// TIA Portal V18 export
// export: Created 2026-03-12T16:04:32.2344065Z, ExportSetting WithDefaults, DisplayName Totally Integrated Automation Portal, DisplayVersion V18 Update 5, DisplayName TIA Portal Openness, DisplayVersion V18 Update 5, DisplayName TIA Portal Version Control Interface, DisplayVersion V18, DisplayName SINAMICS Startdrive Advanced, DisplayVersion V18, DisplayName SINAMICS Startdrive G130, G150, S120, S150, SINAMICS MV, S210, DisplayVersion V18, DisplayName SINAMICS Startdrive G110M, G120, G120C, G120D, G120P, G115D, DisplayVersion V18, DisplayName STEP 7 Professional, DisplayVersion V18 Update 5, DisplayName STEP 7 Safety, DisplayVersion V18, DisplayName WinCC Professional, DisplayVersion V18 Update 5
ORGANIZATION_BLOCK "Main"   // OB1, LAD, ProgramCycle
TITLE = "Main Program Sweep (Cycle)"
{ S7_Optimized_Access := 'TRUE' }
VERSION : 0.1
// Este bloco verifica as condições dos sinais discretos dos painéis. Se as condições operacionais não forem atendidas, as FCs respectivas de cada painel são intertravadas no item 2. Fluxo de Controle.
// stored: AutoNumber true, IsIECCheckEnabled false, SetENOAutomatically false
   VAR_INPUT
      Initial_Call : Bool;   // Initial call of this OB
      Remanence : Bool;   // =True, if remanent data are available
   END_VAR
BEGIN

REGION Network 1: Intertravamento Painel CCO
   // Se o Botão de Emergência estiver Desacionado Painel CCO OK
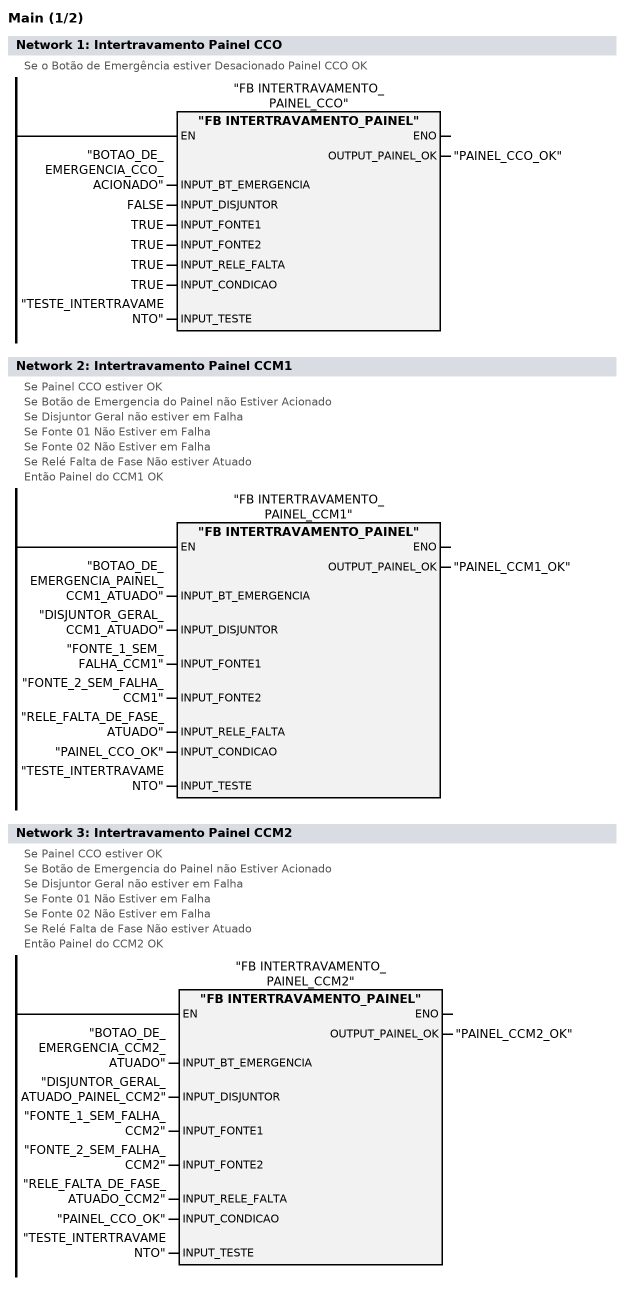
   RUNG wire#powerrail
      "FB INTERTRAVAMENTO_PAINEL_CCO"(INPUT_BT_EMERGENCIA := "BOTAO_DE_EMERGENCIA_CCO_ACIONADO", INPUT_DISJUNTOR := FALSE, INPUT_FONTE1 := TRUE, INPUT_FONTE2 := TRUE, INPUT_RELE_FALTA := TRUE, INPUT_CONDICAO := TRUE, INPUT_TESTE := "TESTE_INTERTRAVAMENTO", OUTPUT_PAINEL_OK => "PAINEL_CCO_OK")
   END_RUNG
   // the same network as SCL:
   "FB INTERTRAVAMENTO_PAINEL_CCO"(INPUT_BT_EMERGENCIA := "BOTAO_DE_EMERGENCIA_CCO_ACIONADO",   // "FB INTERTRAVAMENTO_PAINEL"
                           INPUT_DISJUNTOR := FALSE,
                           INPUT_FONTE1 := TRUE,
                           INPUT_FONTE2 := TRUE,
                           INPUT_RELE_FALTA := TRUE,
                           INPUT_CONDICAO := TRUE,
                           INPUT_TESTE := "TESTE_INTERTRAVAMENTO",
                           OUTPUT_PAINEL_OK => "PAINEL_CCO_OK");
END_REGION

REGION Network 2: Intertravamento Painel CCM1
   // Se Painel CCO estiver OK
   // Se Botão de Emergencia do Painel não Estiver Acionado
   // Se Disjuntor Geral não estiver em Falha
   // Se Fonte 01 Não Estiver em Falha
   // Se Fonte 02 Não Estiver em Falha
   // Se Relé Falta de Fase Não estiver Atuado
   // Então Painel do CCM1 OK
   RUNG wire#powerrail
      "FB INTERTRAVAMENTO_PAINEL_CCM1"(INPUT_BT_EMERGENCIA := "BOTAO_DE_EMERGENCIA_PAINEL_CCM1_ATUADO", INPUT_DISJUNTOR := "DISJUNTOR_GERAL_CCM1_ATUADO", INPUT_FONTE1 := "FONTE_1_SEM_ FALHA_CCM1", INPUT_FONTE2 := "FONTE_2_SEM_FALHA_CCM1", INPUT_RELE_FALTA := "RELE_FALTA_DE_FASE_ATUADO", INPUT_CONDICAO := "PAINEL_CCO_OK", INPUT_TESTE := "TESTE_INTERTRAVAMENTO", OUTPUT_PAINEL_OK => "PAINEL_CCM1_OK")
   END_RUNG
   // the same network as SCL:
   "FB INTERTRAVAMENTO_PAINEL_CCM1"(INPUT_BT_EMERGENCIA := "BOTAO_DE_EMERGENCIA_PAINEL_CCM1_ATUADO",   // "FB INTERTRAVAMENTO_PAINEL"
                           INPUT_DISJUNTOR := "DISJUNTOR_GERAL_CCM1_ATUADO",
                           INPUT_FONTE1 := "FONTE_1_SEM_ FALHA_CCM1",
                           INPUT_FONTE2 := "FONTE_2_SEM_FALHA_CCM1",
                           INPUT_RELE_FALTA := "RELE_FALTA_DE_FASE_ATUADO",
                           INPUT_CONDICAO := "PAINEL_CCO_OK",
                           INPUT_TESTE := "TESTE_INTERTRAVAMENTO",
                           OUTPUT_PAINEL_OK => "PAINEL_CCM1_OK");
END_REGION

REGION Network 3: Intertravamento Painel CCM2
   // Se Painel CCO estiver OK
   // Se Botão de Emergencia do Painel não Estiver Acionado
   // Se Disjuntor Geral não estiver em Falha
   // Se Fonte 01 Não Estiver em Falha
   // Se Fonte 02 Não Estiver em Falha
   // Se Relé Falta de Fase Não estiver Atuado
   // Então Painel do CCM2 OK
   RUNG wire#powerrail
      "FB INTERTRAVAMENTO_PAINEL_CCM2"(INPUT_BT_EMERGENCIA := "BOTAO_DE_EMERGENCIA_CCM2_ATUADO", INPUT_DISJUNTOR := "DISJUNTOR_GERAL_ATUADO_PAINEL_CCM2", INPUT_FONTE1 := "FONTE_1_SEM_FALHA_CCM2", INPUT_FONTE2 := "FONTE_2_SEM_FALHA_CCM2", INPUT_RELE_FALTA := "RELE_FALTA_DE_FASE_ATUADO_CCM2", INPUT_CONDICAO := "PAINEL_CCO_OK", INPUT_TESTE := "TESTE_INTERTRAVAMENTO", OUTPUT_PAINEL_OK => "PAINEL_CCM2_OK")
   END_RUNG
   // the same network as SCL:
   "FB INTERTRAVAMENTO_PAINEL_CCM2"(INPUT_BT_EMERGENCIA := "BOTAO_DE_EMERGENCIA_CCM2_ATUADO",   // "FB INTERTRAVAMENTO_PAINEL"
                           INPUT_DISJUNTOR := "DISJUNTOR_GERAL_ATUADO_PAINEL_CCM2",
                           INPUT_FONTE1 := "FONTE_1_SEM_FALHA_CCM2",
                           INPUT_FONTE2 := "FONTE_2_SEM_FALHA_CCM2",
                           INPUT_RELE_FALTA := "RELE_FALTA_DE_FASE_ATUADO_CCM2",
                           INPUT_CONDICAO := "PAINEL_CCO_OK",
                           INPUT_TESTE := "TESTE_INTERTRAVAMENTO",
                           OUTPUT_PAINEL_OK => "PAINEL_CCM2_OK");
END_REGION

REGION Network 4: Intertravamento Painel CCM3
   // Se Painel CCO estiver OK
   // Se Botão de Emergencia do Painel não Estiver Acionado
   // Se Disjuntor Geral não estiver em Falha
   // Se Fonte 01 Não Estiver em Falha
   // Se Fonte 02 Não Estiver em Falha
   // Se Relé Falta de Fase Não estiver Atuado
   // Então Painel do CCM1 OK
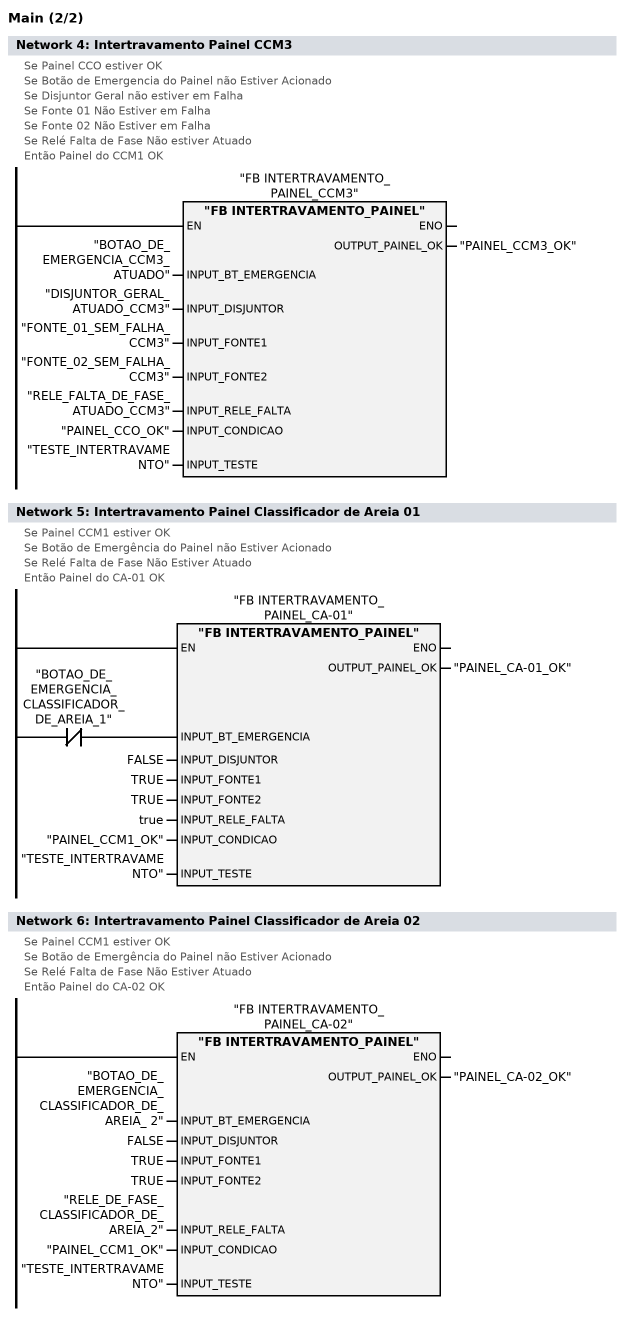
   RUNG wire#powerrail
      "FB INTERTRAVAMENTO_PAINEL_CCM3"(INPUT_BT_EMERGENCIA := "BOTAO_DE_EMERGENCIA_CCM3_ATUADO", INPUT_DISJUNTOR := "DISJUNTOR_GERAL_ATUADO_CCM3", INPUT_FONTE1 := "FONTE_01_SEM_FALHA_CCM3", INPUT_FONTE2 := "FONTE_02_SEM_FALHA_CCM3", INPUT_RELE_FALTA := "RELE_FALTA_DE_FASE_ATUADO_CCM3", INPUT_CONDICAO := "PAINEL_CCO_OK", INPUT_TESTE := "TESTE_INTERTRAVAMENTO", OUTPUT_PAINEL_OK => "PAINEL_CCM3_OK")
   END_RUNG
   // the same network as SCL:
   "FB INTERTRAVAMENTO_PAINEL_CCM3"(INPUT_BT_EMERGENCIA := "BOTAO_DE_EMERGENCIA_CCM3_ATUADO",   // "FB INTERTRAVAMENTO_PAINEL"
                           INPUT_DISJUNTOR := "DISJUNTOR_GERAL_ATUADO_CCM3",
                           INPUT_FONTE1 := "FONTE_01_SEM_FALHA_CCM3",
                           INPUT_FONTE2 := "FONTE_02_SEM_FALHA_CCM3",
                           INPUT_RELE_FALTA := "RELE_FALTA_DE_FASE_ATUADO_CCM3",
                           INPUT_CONDICAO := "PAINEL_CCO_OK",
                           INPUT_TESTE := "TESTE_INTERTRAVAMENTO",
                           OUTPUT_PAINEL_OK => "PAINEL_CCM3_OK");
END_REGION

REGION Network 5: Intertravamento Painel Classificador de Areia 01
   // Se Painel CCM1 estiver OK 
   // Se Botão de Emergência do Painel não Estiver Acionado
   // Se Relé Falta de Fase Não Estiver Atuado 
   // Então Painel do CA-01 OK
   RUNG wire#powerrail
      "FB INTERTRAVAMENTO_PAINEL_CA-01"(INPUT_BT_EMERGENCIA := wire#w1, INPUT_DISJUNTOR := FALSE, INPUT_FONTE1 := TRUE, INPUT_FONTE2 := TRUE, INPUT_RELE_FALTA := true, INPUT_CONDICAO := "PAINEL_CCM1_OK", INPUT_TESTE := "TESTE_INTERTRAVAMENTO", OUTPUT_PAINEL_OK => "PAINEL_CA-01_OK")
   END_RUNG
   RUNG wire#powerrail
      I_Contact( "BOTAO_DE_EMERGENCIA_CLASSIFICADOR_DE_AREIA_1" )
   END_RUNG wire#w1
   // the same network as SCL:
   "FB INTERTRAVAMENTO_PAINEL_CA-01"(INPUT_BT_EMERGENCIA := NOT "BOTAO_DE_EMERGENCIA_CLASSIFICADOR_DE_AREIA_1",   // "FB INTERTRAVAMENTO_PAINEL"
                           INPUT_DISJUNTOR := FALSE,
                           INPUT_FONTE1 := TRUE,
                           INPUT_FONTE2 := TRUE,
                           INPUT_RELE_FALTA := true,
                           INPUT_CONDICAO := "PAINEL_CCM1_OK",
                           INPUT_TESTE := "TESTE_INTERTRAVAMENTO",
                           OUTPUT_PAINEL_OK => "PAINEL_CA-01_OK");
END_REGION

REGION Network 6: Intertravamento Painel Classificador de Areia 02
   // Se Painel CCM1 estiver OK 
   // Se Botão de Emergência do Painel não Estiver Acionado
   // Se Relé Falta de Fase Não Estiver Atuado 
   // Então Painel do CA-02 OK
   RUNG wire#powerrail
      "FB INTERTRAVAMENTO_PAINEL_CA-02"(INPUT_BT_EMERGENCIA := "BOTAO_DE_EMERGENCIA_CLASSIFICADOR_DE_AREIA_ 2", INPUT_DISJUNTOR := FALSE, INPUT_FONTE1 := TRUE, INPUT_FONTE2 := TRUE, INPUT_RELE_FALTA := "RELE_DE_FASE_CLASSIFICADOR_DE_AREIA_2", INPUT_CONDICAO := "PAINEL_CCM1_OK", INPUT_TESTE := "TESTE_INTERTRAVAMENTO", OUTPUT_PAINEL_OK => "PAINEL_CA-02_OK")
   END_RUNG
   // the same network as SCL:
   "FB INTERTRAVAMENTO_PAINEL_CA-02"(INPUT_BT_EMERGENCIA := "BOTAO_DE_EMERGENCIA_CLASSIFICADOR_DE_AREIA_ 2",   // "FB INTERTRAVAMENTO_PAINEL"
                           INPUT_DISJUNTOR := FALSE,
                           INPUT_FONTE1 := TRUE,
                           INPUT_FONTE2 := TRUE,
                           INPUT_RELE_FALTA := "RELE_DE_FASE_CLASSIFICADOR_DE_AREIA_2",
                           INPUT_CONDICAO := "PAINEL_CCM1_OK",
                           INPUT_TESTE := "TESTE_INTERTRAVAMENTO",
                           OUTPUT_PAINEL_OK => "PAINEL_CA-02_OK");
END_REGION

REGION Network 7: Comunicação Supervisório
END_REGION
END_ORGANIZATION_BLOCK
